{attribute addProperty BoxType "EK1100-0000-0018"}
{attribute addProperty Id "Beckhoff_EL15xxEK1122Beckhoff_EL15xxEK1122_50B385EA162A_0001_EL1502_0000_0000EL1502_BA17F41223429.25A_0002_EL1502_0000_0001EL1502_307D150D24230.25A_0003_EL1502_0000_0016EL1502_307D150D24230.25A_0004_EL1502_0000_0017EL1502_307D150D24230.25A_0005_EL1502_0000_0018EL1502_190A00FC17822.25A_0006_EL1502_0000_0019EL1502_190A00FC17822.25A_0007_EL1502_0000_0020EL1502_190A00FC17822.25A_0008_EL1502_0000_0021EL1502_190A00FC17822.25A_0009_EL1502_0000_0022EL1502_190A00FC17822.25A_0010_EL1512_0000_0016EL1512_736E064C30638.25A_0011_EL1512_0000_0017EL1512_7D86CA5B27434.25A_0012_EL1512_0000_0018EL1512_7D86CA5B27434.25A_0013_EL1512_0000_0019EL1512_7D86CA5B27434.25A_0014_EL1512_0000_0020EL1512_7D86CA5B27434.25A_0015_EL1512_0000_0021EL1512_7D86CA5B27434.25"}
{attribute addProperty CRC "3680105850"}
{attribute addProperty SizeInBites "3542"}
{attribute addProperty SizeInBytes "442.75"}
TYPE Beckhoff_EL15xx_DB59F57A EXTENDS EK1100_179A0949 :
STRUCT
	{attribute addProperty Name "Beckhoff_EL15xxEK1122"}
	Beckhoff_EL15xxEK1122 : Beckhoff_EL15xxEK1122_50B385EA;
	{attribute addProperty Name "A_0001_EL1502_0000_0000"}
	A_0001_EL1502_0000_0000 : EL1502_BA17F412;
	{attribute addProperty Name "A_0002_EL1502_0000_0001"}
	A_0002_EL1502_0000_0001 : EL1502_307D150D;
	{attribute addProperty Name "A_0003_EL1502_0000_0016"}
	A_0003_EL1502_0000_0016 : EL1502_307D150D;
	{attribute addProperty Name "A_0004_EL1502_0000_0017"}
	A_0004_EL1502_0000_0017 : EL1502_307D150D;
	{attribute addProperty Name "A_0005_EL1502_0000_0018"}
	A_0005_EL1502_0000_0018 : EL1502_190A00FC;
	{attribute addProperty Name "A_0006_EL1502_0000_0019"}
	A_0006_EL1502_0000_0019 : EL1502_190A00FC;
	{attribute addProperty Name "A_0007_EL1502_0000_0020"}
	A_0007_EL1502_0000_0020 : EL1502_190A00FC;
	{attribute addProperty Name "A_0008_EL1502_0000_0021"}
	A_0008_EL1502_0000_0021 : EL1502_190A00FC;
	{attribute addProperty Name "A_0009_EL1502_0000_0022"}
	A_0009_EL1502_0000_0022 : EL1502_190A00FC;
	{attribute addProperty Name "A_0010_EL1512_0000_0016"}
	A_0010_EL1512_0000_0016 : EL1512_736E064C;
	{attribute addProperty Name "A_0011_EL1512_0000_0017"}
	A_0011_EL1512_0000_0017 : EL1512_7D86CA5B;
	{attribute addProperty Name "A_0012_EL1512_0000_0018"}
	A_0012_EL1512_0000_0018 : EL1512_7D86CA5B;
	{attribute addProperty Name "A_0013_EL1512_0000_0019"}
	A_0013_EL1512_0000_0019 : EL1512_7D86CA5B;
	{attribute addProperty Name "A_0014_EL1512_0000_0020"}
	A_0014_EL1512_0000_0020 : EL1512_7D86CA5B;
	{attribute addProperty Name "A_0015_EL1512_0000_0021"}
	A_0015_EL1512_0000_0021 : EL1512_7D86CA5B;
END_STRUCT
END_TYPE

(* stored: Version 1.2.0.0, ProductVersion 3.1.4024.9
   DUT Beckhoff_EL15xx_DB59F57A: Id {d626b346-e6cf-43d4-a63e-3b860503b3bd} *)
